FUNCTION_BLOCK BasicObject EXTENDS ITF_Cyclic
VAR_INPUT
END_VAR
VAR_OUTPUT
END_VAR
VAR
END_VAR

END_FUNCTION_BLOCK

(* stored: Version 1.1.0.1, ProductVersion 3.1.4024.12
   POU BasicObject: Id {2033108e-e225-43e0-87bf-73fc6ab5005b}, SpecialFunc None *)
